RESOURCE_TYPE _Core0
  (* Standard: 61499-2 *)
  (* Version 0.1, 2017-00-09, hpea485, UOA *)
  VAR_INPUT
    Core0Input : INT;
  END_VAR
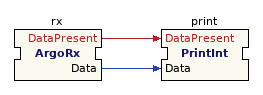
  FBS
    rx : ArgoRx;
    print : PrintInt;
  END_FBS
  EVENT_CONNECTIONS
    rx.DataPresent TO print.DataPresent;
  END_CONNECTIONS
  DATA_CONNECTIONS
    rx.Data TO print.Data;
  END_CONNECTIONS
END_RESOURCE_TYPE
